# B&R Automation Studio project TD52 (part 46)

#### c_spare3Init.st
```iecst
(*******************************************************************************
CUSTOMIZED: c_spare3 			init to customized task placeholder

This code is confidential and proprietary to the INNIO Company.
It may not be used in any form, or reproduced in any manner,
without written permission of the INNIO Company.
Copyright, INNIO Company, 2019

Customized modifications: -
------------------------

Instructions for use:
--------------------
USE THIS TASK TO ADD CODE SNIPPETS AFTER ENGINE DELIVERY

Outstandings:
------------

*******************************************************************************)
PROGRAM _INIT

	bDoNothing := TRUE;

	(*-----------------------------------------------------------------------------*)
	bNoInitDetected := FALSE; 	 (* Insert this into every tasks INIT code to activate download detection *)
END_PROGRAM
```

### Program Logical/Customized/c_mns (IEC, version 4.14.0) - customisation task for grid power controller

#### c_mnsCyclic.st
```iecst
(*******************************************************************************
c_mns		 customizable mains demand controller  (derived from anf_nb 	customized engine demand depending of griddemand power setpoints)

This code is confidential and proprietary to the INNIO Company.
It may not be used in any form, or reproduced in any manner,
without written permission of the INNIO Company.
Copyright, INNIO Company, 2025

Customized modifications: -
------------------------

History:
-------
V4.04.1 14.11.2016 Zengerer			New task according to new spec. from Schwab Christoph, TPE (based on task anf_nb V4.03.0, 05.07.2013 pankayrodney)
V4.04.2 23.05.2017 Zengerer			Connect IN Interfaces to Hal tP_Mns_AnaIn, tDem_Ctr_Mns
V4.05.0 05.09.2017 zengerer			Nachziehen der Netzbezugsregler Änderungen von Schwab Christoph / Caks Michael aus File Bugs&Solution_MnsCtrl.zip
V4.05.1 30.11.2017 zengerer			50 + removed according to Basisupdate 4.4.0.6
V4.05.2 12.03.2018 zengerer			comments updated
V4.05.3 18.04.2018 Schwab Christoph bMsg2302_Enable-- bMsg2418_Enable Version
V4.05.4 20.04.2018 Zengerer			Timer Reset Button FUNCTION INVERTED; SOME UNTESTED CHANGES FROM V4.5.3 REVERTED
		25.04.2018 Zengerer			MM2VIS.rPmns_DemGenerate_Lim_On rPmns_DemGenerate_Lim_Off
V4.07.1 13.05.2019 Zengerer		 	Change of y_Min Y_Max strategy per option selection, ShadowPara_tCtr_Mns to prevent para writing; +activation Para
V4.11.0	24.02.2022 Perktold			impemented plant controller upgrade
V4.14.0	13.03.2025 Zengerer 		moved mains import controller activation bit

Instructions for use:
--------------------
 TASK REPLACES the task anf_nb. Do not activate anf_nb any more.

Outstandings:
------------
ADOPT ACCORDING TO PLANT SPECIFIC NEEDS

	-Testing for IN_CU.tP_Act[2].Ai has to be done
	-remove SparePara[73] V4.07 option here after testing phase
*******************************************************************************)
PROGRAM _CYCLIC

	(* IN INTERFACE: new V4.4.0,  2016 *)
	IN_CU.tDem_Ctr_Mns.Di	;				(*activation bit input (default value in case of not using interface moved to c_modIF) *)
	bDem_Ctr_Mns := IN_CU.tDem_Ctr_Mns.Di;  (*connect DI mns controller activation interface to hardware *)
	IN_CU.tP_Mns_AnaIn.Ai  ; 				(*AnaIn		Mains power Actual value over mA Signal *)
	IN_CU.tP_Mns_AnaIn.GoodQual ;			(*AnaIn		Mains power Actual value over mA Signal *)
	IN_CU.tP_Act[2].Ai;						(* P [kW] 	Mains power Actual value over MMU	*)

	IN_CU.rP_Nom;							(*Nominal power at selected gas type *)

	VIS2MM.tCtr_Mns_In;
//	VIS2MM.rPmns_setpoint ;					(* = p_MainsImport Setpoint *)
	IN_CU.tCtr_Mns_Anain_Setp_W_ext.Ai;		 (*AnaIn	Setpoint over mA Signal *)	//replaces:  = 	OUT_CU.rCustAnaIn[1] /100.0 ;
	IN_CU.tCtr_Mns_Anain_Setp_W_ext.GoodQual;(*AnaIn	Setpoint over mA Signal *)	//replaces:  = 	OUT_CU.rCustAnaIn[1] /100.0 ;

	Para.bCtr_Mns_Enable;				(*Parameter)	general activation bit for mns controller *)

	Para.tCtr_Mns.W_set;				(*Parameter	W(setpoint) start  Var.1:	internal setpoint *)
	Para.tCtr_Mns.W_min;				(*Parameter	W(setpoint) minimum *)
	Para.tCtr_Mns.W_max;				(*Parameter	W(setpoint) maximum *)
	Para.bCtr_Mns_AnaIn_Setp_Enable;	(*Parameter 	setpoint over mA aktiv Var.2: analog in setpoint *)
	Para.bCtr_Mns_Setp_Set4mA;			(*Parameter 	scaling 4-20 mA aktiv *)
	Para.rCtr_Mns_Setp_ScalMin;			(*Parameter 	scale minimum *)
	Para.rCtr_Mns_Setp_ScalMax;			(*Parameter 	scale maximum *)

	Para.bP_Mns_MMU_Enable;				(*Parameter 	TRUE = use MMU2 measurement reading, FALSE = use Analog Input reading from customer messurement euipment *)
	Para.bP_Mns_AnaIn_Enable := NOT Para.bP_Mns_MMU_Enable;		(*INTERNAL GENERATED HERE, necessary because bP_Mns_AnaIn_Enable is not a parameter on VIS anymore*)

	Para.bP_Mns_AnaIn_Set4mA;			(*Parameter 	value scaling 4-20 mA aktiv *)
	Para.rP_Mns_AnaIn_ScalMin;			(*Parameter 	scale minimum *)
	Para.rP_Mns_AnaIn_ScalMax;			(*Parameter 	scale maximum *)

	Para.bLimOnOff_aktiv;				(*Parameter)	TRUE = use mns-ctr output to perform engine demand on/off *)
	Para.rMainsImport_max;				(*Parameter)	Mains Import maximum warning limit	*)
	Para.rMainsImport_max_trip;			(*Parameter)	Mains Import maximum alarm limit *)
	Para.rMainsExport_max;				(*Parameter)	Mains Export maximum warning limit	*)
	Para.rMainsExport_max_trip;			(*Parameter)	Mains Export maximum alarm limit *)

	Para.rDemGenerate_Lim_On;			(*Parameter)	Grenzwert Einschaltung (% von PN Generator) *)
	Para.rTime_Dem_On_delay;			(*Parameter)	Delay time until engine demand on [sec] *)
	Para.rDemGenerate_Lim_Off;			(*Parameter)	Grenzwert Abschaltung (% von PN Generator) *)
	Para.rTime_Dem_Off_delay;			(*Parameter)	Delay time until engine demand off [sec]*)
	Para.tCtr_Mns.W_set;				(*Parameter)	W(setpoint) start *)

	(* OUT INTERFACE *)
	OUT_CU.bEngDSS_Mains  ;								(* == ANF_NB *)
	OUT_CU.rP_MainsImport ;				(* rP_MainsImport Interface to MM syncronising: +=grid to plant power value in [KW] *)
	OUT_CU.rP_Set_Mns_Norm;				(* engine power setpoint from grid controller out   *)

	MM2VIS.bEngDSS_Mains ;	// := OUT_CU.bEngDSS_Mains;	(* == ANF_NB *)
	MM2VIS.rPcsm_act ;					(* Consumer Power = p_MainsImport + rP_Act_Norm_Filt *)
	MM2VIS.rPmns_act ;		//:= OUT_CU.rP_MainsImport ;					(* p_MainsImport t (= OUT_CU.rP_MainsImpor) *)
	MM2VIS.rPmns_setpoint ;				(* selected p_MainsImport Setpoint, with ramps... *)
	MM2VIS.tCtr_Mns_Out;				(*Controler output structure for VIS*)
	MM2VIS.tCtr_Mns_Out.Active;			(*Controler output active*)
	MM2VIS.tCtr_Mns_Out.Y;				(* engine power etpoint from grid controller out   *)

	OUT_CU.tCtr_Mns_Out ;				(*Controler output structure *)
	OUT_CU.tCtr_Mns_In;					(*Copy of controler input structure for reuse in other modules *)

	(****************************************************************************************************)
	(*Calculation of power values*)
	//Mains Power set point import controller
	IF 	(*Para.bP_Mns_AnaIn_Enable*)Para.bCtr_Mns_AnaIn_Setp_Enable  AND IN_CU.tCtr_Mns_Anain_Setp_W_ext.GoodQual THEN // Schwab Ch. Falscher Parameter Angebunden	(*Parameter setpoint over mA aktiv Var.2:	Der Sollwert wird mittels externen mA Signal, welches über Parameter angepasst werden kann*)
		rP_Mains_Set := IN_CU.tCtr_Mns_Anain_Setp_W_ext.Ai;		(*AnaIn		Setpoint over mA Signal *)

	ELSE
	//	rP_Mains_Set := MM2VIS.tCtr_Mns_Out.W;			NEIN, GEHT hier SO NICHT mehr!	(* rP_GenerateSet		alt: 	soll_netz := REG1.w;*)
		rP_Mains_Set := Para.tCtr_Mns.W_set;  		(* rP_GenerateSet from Vis manual input	*)
	END_IF

	//Verbraucherleistung (= Netzbezugsleistung + Generatorleistung)
	rP_Consumption := rP_MainsImport + (IN_CU.rP_Act_Norm_Filt * IN_CU.rP_Nom);			(* verbrauch == rP_Consumption					alt: verbrauch := netzbezug + );*)

	(*Schwab Ch. => rP_DemGenerate wird immer berechnet! Keine IF Funktion benötigt*)
	rP_DemGenerate := rP_Consumption - rP_Mains_Set;
	MM2VIS.rPmns_DemGenerate := rP_DemGenerate;		(*new V4.5 beta *)

	(* P_MainsImport: measured absolute power from mains to plant in [KW] (+=grid to plant power, -=plant to grid*)	 //=Netzbezugsleistung
	IF 	Para.bP_Mns_MMU_Enable THEN 							(*Parameter TRUE = ISTwert Netzbezug über MMU gemessen (Var.2), 	FALSE = über mA Signal (Var.1)*)
		//FEHLT NOCH: NB- Leistung von eigenem MMU
		rP_MainsImport := 	IN_CU.tP_Act[2].Ai;					(* P [kW] Mains power Actual value over MMU	  := 98765.4321;		//FEHLT NOCH:  test  *)

	ELSIF  IN_CU.tP_Mns_AnaIn.GoodQual THEN 				(*AnaIn	Actual value mA Signal Quality Check*)
		rP_MainsImport := 	IN_CU.tP_Mns_AnaIn.Ai;		(*AnaIn	Istwert = über mA Signal (Var.1):	Der Istwert wird mittels mA Signal geliefert, welches über Parameter angepasst werden kann	 	alt: netzbezug := REAL_TO_INT(OUT_CU.rCustAnaIn[1]);	*)
	ELSE
		rP_MainsImport :=	(-rP_MainsImport_max) ;				(* failsafe value = no engine demand *)
	END_IF

	IF 	Para.bCtr_Mns_Enable AND bDem_Ctr_Mns THEN 	 (* TASK ACTIVATION by (Parameter)	Regler Aktivierung *)

		(* P_MainsImport_max limit parameter*)	//maximal erlaubte Netzbezugsleistung
	//	rP_MainsImport_max := DINT_TO_REAL(Para.rCust_SparePara[1]);		(*:= SPS_REZP1;				alt:netzbezug_max := INT_TO_UDINT(Para.rCust_SparePara[1]); *)
		rP_MainsImport_max :=  			Para.rMainsImport_max;				(*Parameter)	Mains Import maximum	alt:netzbezug_max := INT_TO_UDINT(Para.rCust_SparePara[1]); *)
						// old:			Para.rMainsImport_max_trip;			(*Parameter)	Mains Import maximum Abstellend True/False *)

		//Grenzwert [0-1 NOM Pnenn (früher %Pnenn!)] Anforderung EIN
		rP_DemGenerate_Lim_On :=		Para.rDemGenerate_Lim_On;			(*Parameter)	Grenzwert Einschaltung (% von PN Generator)  alt: p_ein_proz := INT_TO_UDINT( SPS_REZP1); *)

		//Grenzwert [0-1 NOM Pnenn (früher %Pnenn!)] Anforderung AUS
		rP_DemGenerate_Lim_Off :=		Para.rDemGenerate_Lim_Off;			(*Parameter)	Grenzwert Abschaltung (% von PN Generator) 	alt: p_aus_proz := INT_TO_UDINT( SPS_REZP2);*)

		//Nennleistung bei aktiver Gasart
		rP_Nom := (IN_CU.rP_Nom);					(*Nennleistung bei aktiver Gasart)  alt: zm := REAL_TO_INT(IN_CU.P_Nom);*)

		//Freigabe Netzbezugsregler
		//bDem_Ctr_Mns :=  ?  := bRSS_Rem AND IN_CU.bMCB_On AND IN_CU.GCB_ON AND IN_CU.AN_PGW1;		(*kann bRSS_Rem ersetzt werden durch bRSS_Rem? - nein *)
		OUT_CU.bEngDSS_Mains_Rel := IN_CU.bOMSS_Aut
								AND bRSS_Rem
								AND	IN_CU.bMCB_On
								AND Para.bCtr_Mns_Enable
								//	IN_CU.bGCB_On AND  NICHT einbinden, Regler kann sonst den motor nicht mehr starten!
								AND bDem_Ctr_Mns 	(*DI Customer Demand Input*)
								AND	(IN_CU.tP_Mns_AnaIn.GoodQual OR IN_CU.tP_Act[2].GoodQual);		(*lt. Schwab, 2017-11-28*)

		(*OUT_CU.bEngDSS_Mains_Block aktuell nicht in Verwendung => Wird über A2302 abgedeckt /  Schwab Ch.*)
		//		//Notabschaltung durch Überschreitung der erlaubten Rückspeiseleistung ins Netz (pb7/M_BLOCK)
//		xTOF_FA_BLOCK_NB.IN := (-rP_MainsImport) > rP_MainsImport_max;				(*shut down engine, if power to grid (=-MainsImport) exceeds allowed limt *)
//		xTOF_FA_BLOCK_NB.PT := REAL_TO_TIME(Para.rTime_Dem_Off_delay) * 1000;			(*Parameter)	[SEC] Zeitwert Verzögerung Abforderung alt: T#1m; *)
//		xTOF_FA_BLOCK_NB();
//
//		OUT_CU.bEngDSS_Mains_Block := xTOF_FA_BLOCK_NB.Q;

		//geforderte Generatorleistung (= Verbraucherleistung - Netzbezugsollwert)
//		IF bDem_Ctr_Mns THEN
//			rP_DemGenerate := MM2VIS.tCtr_Mns_Out.Y * rP_Nom; //Funktion doppelt? ->sonst TESTEN!
//		ELSE
//			rP_DemGenerate := rP_Consumption - rP_Mains_Set;					(*	soll_gen ==  rP_DemGenerate		alt: soll_gen := verbrauch - soll_netz; *)
//		END_IF

		//Berechnung Anforderungsleistung
//		zm1 := rP_DemGenerate_Lim_On * rP_Nom;				//Schwab remove: 50 + rP_DemGenerate_Lim_On * rP_Nom
////	zm1 := zm1/100;
//		p_ein := (zm1);												(*UDINT_TO_INT(zm1);*)
		p_ein := rP_DemGenerate_Lim_On * rP_Nom;			//Schwab remove: 50 + rP_DemGenerate_Lim_On * rP_Nom
		MM2VIS.rPmns_DemGenerate_Lim_On := p_ein;		(*new V4.5 beta *)

		//Berechnung Abwahlleistung
//		zm0 := rP_DemGenerate_Lim_Off * rP_Nom;				//Schwab remove: 50 + rP_DemGenerate_Lim_Off * rP_Nom
////	zm0 := zm0/100;
//		p_aus := (zm0);												(*UDINT_TO_INT(zm0);*)
		p_aus := rP_DemGenerate_Lim_Off * rP_Nom;			//Schwab remove: 50 + rP_DemGenerate_Lim_Off * rP_Nom
		MM2VIS.rPmns_DemGenerate_Lim_Off := p_aus;		(*new V4. beta5 *)

		//Anforderung EIN
		IF AUS AND NOT bDisplayTimerHelper THEN
			TON_R_MnsDemandOn.PT := REAL_TO_UDINT(Para.rTime_Dem_On_delay) * 100;
		END_IF
		TON_R_MnsDemandOn(IN := (rP_DemGenerate >= p_ein));				(*caution, RS will NOT WORK here as intended! *)
	//	TON_R_MnsDemandOn(IN := (rP_DemGenerate >= p_ein), PT := 	(Para.tiTime_Dem_On_delay) * 1000, RS := VIS2MM.bTime_Dem_On_delay_Reset);
		IF VIS2MM.bTime_Dem_On_delay_Reset	THEN		(*IF VIS Timer Reset Button is pressed*)
			VIS2MM.bTime_Dem_On_delay_Reset := FALSE;	(*clear button*)
			TON_R_MnsDemandOn( PT := 0 );				(*runout timer*)
			TON_R_MnsDemandOff( PT := 0 );				(*runout timer*)
			bDisplayTimerHelper := TRUE;				(*Visu helper bit for TON_R_MnsDemandOn display*)
		END_IF
		IF (IN_CU.rN_EngAct > 450) AND (IN_CU.rN_EngAct < 750) THEN 	bDisplayTimerHelper := FALSE; END_IF			(*Reset Visu helper bit for TON_R_MnsDemandOn display*)

		EIN := TON_R_MnsDemandOn.Q;
		MM2VIS.rTime_Dem_On_CntDn := UDINT_TO_REAL(TON_R_MnsDemandOn.PT - TON_R_MnsDemandOn.ET) /100 ;		(* Display start count down *)
	//	MM2VIS.tiTime_Dem_On_CntDn := 			  (TON_R_MnsDemandOn.PT - TON_R_MnsDemandOn.ET) /1000 ;		(* Display start count down *)

		//Anforderung AUS
		IF EIN AND NOT bDisplayTimerHelper THEN
			TON_R_MnsDemandOff.PT := REAL_TO_UDINT(Para.rTime_Dem_Off_delay) * 100; 	(*Parameter)	Delay time until engine demand off [sec]*)
			MM2VIS.rTime_Dem_On_CntDn := UDINT_TO_REAL(TON_R_MnsDemandOff.PT - TON_R_MnsDemandOff.ET) /100 ;		(* Display start count down *)
		END_IF
		TON_R_MnsDemandOff(IN := (rP_DemGenerate <= p_aus));		(* PREPARED for AUS := soll_gen <= p_aus;*)
		AUS := 	TON_R_MnsDemandOff.Q;
	//	AUS := rP_DemGenerate <= p_aus;								(* := soll_gen <= p_aus;*)

		//Anforderung
		OUT_CU.bEngDSS_Mains := (EIN OR OUT_CU.bEngDSS_Mains)
							AND NOT AUS			(* OUT_CU.bEngDSS_Mains == ANF_NB *)
							AND Para.bLimOnOff_aktiv;

		(*Connection failure bit for message set*)
		(* A2302 mains export power limit: Shut down engine, if NEGATIVE Mains Import (= power export to the grid) is exceeding (<) the allowed limit (-Limit value)  *)
		bMsg2302_Enable	:=	Para.bCtr_Mns_Enable
//						AND Para.bLimOnOff_aktiv 				// gehört nicht zu dieser Funktion / Schwab Ch.
						AND ((*IN_CU.tDem_Ctr_Mns.Di*)bDem_Ctr_Mns OR Para.iCtr_Mns_Options.2);

		bMsg2302_Set	:=	OUT_CU.rP_MainsImport < (-Para.rMainsExport_max_trip);

		(* A2303 mains import controller limit 2  ??? Why shut down the engine, if too few power is available  ???	*)
		bMsg2303_Enable	:=	Para.bCtr_Mns_Enable
//						AND Para.bLimOnOff_aktiv 				// gehört nicht zu dieser Funktion / Schwab Ch.						AND Para.bLimOnOff_aktiv
						AND (*IN_CU.tDem_Ctr_Mns.Di*)bDem_Ctr_Mns
						AND ((*IN_CU.tDem_Ctr_Mns.Di*)bDem_Ctr_Mns OR Para.iCtr_Mns_Options.3) 			(*Change 2018 Ze: Alarm only active in Ctr_Mns mode (using option bit 3 and 4 of INTERNAL parameter, ->NORMALY SWITCHED TO FALSE*)
						AND Para.iCtr_Mns_Options.4
						AND FALSE;	// Funktion muss nochmals mit betroffene Personen diskutiert werden / Schwab Ch.

		bMsg2303_Set	:= OUT_CU.rP_MainsImport > Para.rMainsImport_max_trip;

		(* W2415 mains import controller: Messsignalstörung Netzbezugs- Sollwert 	*)
		bMsg2415_Enable	:=	Para.bCtr_Mns_Enable
						AND Para.bCtr_Mns_AnaIn_Setp_Enable
						AND (IN_CU.tDem_Ctr_Mns.Di OR Para.iCtr_Mns_Options.5);	(*Change 2018 Ze: Alarm only active in Ctr_Mns mode (using option bit 5 and 4 of INTERNAL parameter, ->NORMALY SWITCHED TO FALSE*)

		bMsg2415_Set	:= NOT IN_CU.tCtr_Mns_Anain_Setp_W_ext.GoodQual;

		(* W2416 mains import controller: Messsignalstörung Netzbezugs- Istwert	*)
		bMsg2416_Enable	:=	Para.bCtr_Mns_Enable
						AND	bDem_Ctr_Mns
						AND Para.bP_Mns_AnaIn_Enable
						AND Para.bP_Mns_AnaIn_Set4mA
						AND ((*IN_CU.tDem_Ctr_Mns.Di*)bDem_Ctr_Mns OR (NOT Para.iCtr_Mns_Options.6));

		bMsg2416_Set	:= NOT IN_CU.tP_Mns_AnaIn.GoodQual;

		(* W2417 mains export power limit: Warning, if NEGATIVE Mains Import (= power export to the grid) is exceeding (<) the allowed limit (-Limit value)  *)
		bMsg2417_Enable	:=	Para.bCtr_Mns_Enable  					//AND Para.bLimOnOff_aktiv;
						AND bDem_Ctr_Mns
						AND ((*IN_CU.tDem_Ctr_Mns.Di*)bDem_Ctr_Mns OR (NOT Para.iCtr_Mns_Options.7));

		bMsg2417_Set	:= OUT_CU.rP_MainsImport < (-Para.rMainsExport_max) ;

		(* W2418  mains import controller limit 2:  Warning if positive Mains Import (= power drawn from the grid) is exceeding (>) the allowed limit (+Limit value)*)
		bMsg2418_Enable	:=	Para.bCtr_Mns_Enable 					//AND Para.bLimOnOff_aktiv AND FALSE;
						AND bDem_Ctr_Mns
						AND ((*IN_CU.tDem_Ctr_Mns.Di*) bDem_Ctr_Mns OR Para.iCtr_Mns_Options.8);

		bMsg2418_Set	:= OUT_CU.rP_MainsImport > Para.rMainsImport_max;

	ELSE
		//Task disabeled, keine Anforderung
		bMsg2302_Enable		 		:= FALSE;
		bMsg2302_Set		 		:= FALSE;
		bMsg2303_Enable		 		:= FALSE;
		bMsg2303_Set		 		:= FALSE;
		bMsg2415_Enable		 		:= FALSE;
		bMsg2415_Set		 		:= FALSE;
		bMsg2416_Enable		 		:= FALSE;
		bMsg2416_Set		 		:= FALSE;
		bMsg2417_Enable		 		:= FALSE;
		bMsg2417_Set		 		:= FALSE;
		bMsg2418_Enable		 		:= FALSE;
		bMsg2418_Set		 		:= FALSE;
		OUT_CU.bEngDSS_Mains 		:= FALSE;
		OUT_CU.bEngDSS_Mains_Rel	:= FALSE;

	END_IF

	(******************************************************************************)
	(* MAINS POWER IMPORT/EXPORT CONTROLLER [kW] (System 1 from Lettenbichler- Plant Control) *)
//	IF 	Para.bCtr_Mns_Enable  THEN 	 (* ACTIVATION by (Parameter)  V4.07:  integratet in .enable *)
		(* PlantOperMode = 1 *)
		VIS2MM.tCtr_Mns_In.enable   	:= 	OUT_CU.bEngDSS_Mains_Rel AND Para.bCtr_Mns_Enable ; //bDem_Ctr_Mns ;		(*(Schnittstelle)	Aktivierung über Kundenschnittstelle *)
		VIS2MM.tCtr_Mns_In.W_ext    	:=  rP_Mains_Set;  				(*	Setpoint over mA Signal  FEHLT NOCH: .w_ref    := MAX (IN_MC.ENG_nom[1].Pgen, Pgen_dmnd_nom);(* reference value, units like "x" *)
		VIS2MM.tCtr_Mns_In.W_ext_Active := 	Para.bCtr_Mns_AnaIn_Setp_Enable ;		(* setpoint activation,  old: Para.Pmns_sp;  *)

		VIS2MM.tCtr_Mns_In.W_set2_Active	:= FALSE;	(*Input to define which internal setpoint will be used TRUE = use the 2nd set point | FALSE use the normal "1st" one*)
		VIS2MM.tCtr_Mns_In.GainScheduling	:= 0.0;		(*Input for Gain Scheduling: 0.0 = use 100% of the Standard PID-Parameters | 1.0 = use 100% of the GainSched. PID Parameters | linear interpolation in between*)
		VIS2MM.tCtr_Mns_In.Y_min_cust;					(*"customized" Y-Min at the current moment (The existing Y-Min parameter is the global minimum. To have an effect Y_min_cust needs to be > the parameter | -1.0 = function not used*)
		VIS2MM.tCtr_Mns_In.Y_max_cust;					(*"customized" Y-Max at the current moment (The existing Y-Max parameter is the global maximum. To have an effect Y_max_cust needs to be < the parameter | 1.0 = function not used*)
		VIS2MM.tCtr_Mns_In.Retrigger;					(*a rising edge on this input signals the controller to retrigger - set W on X and force the Integrator to the current Y*)
		VIS2MM.tCtr_Mns_In.A;							(*feed forward Input*)

		VIS2MM.tCtr_Mns_In.X			:= rP_MainsImport;				(* actual value, "PV Name" of "x" *)

		//	VIS2MM.tCtr_Mns_In.mode     	:= 1;   	     		     	(* 1: dy=Ki*(w-x/w_ref), 0: dy=Ki *)

		Para.tCtr_Mns.deadband	;  // 	:= 10.0;				(* dead band, units like "x" *)
		IF Para.tCtr_Mns.Tn = 0 THEN Para.tCtr_Mns.Tn := 110; END_IF // VIS2MM.tCtr_Mns_In.Ki_plus  := Speed_P_Ad/10;	(* units "In"/100ms=task class *)
									 Para.tCtr_Mns.Tn  ; 			 // VIS2MM.tCtr_Mns_In.Ki_minus := Speed_P_Ad/10;	(* units "In"/100ms=task class *)
		IF Para.tCtr_Mns.dY_max = 0 THEN Para.tCtr_Mns.dY_max := 0.1;	END_IF			(*  *)
		Para.tCtr_Mns.Y_block  	;	//:= 1.0;				(* % *)

		Para.tCtr_Mns.invert   ; 		//  := TRUE;			 	(* FALSE: x>w: decrease y, TRUE: x>w: increase y *)

		(*Beginn V4.07 change *)
		ShadowPara_tCtr_Mns			:= Para.tCtr_Mns;	(* controler internal derouting of para *)

		rY_min	:= LIMIT( (IN_CU.rP_Act_Norm_Filt - 0.03), (IN_CU.rP_Set_Min_Norm -0.03), 1.0);
		rY_max	:= LIMIT( (IN_CU.rP_Act_Norm_Filt + 0.03),  IN_CU.rP_Set_Min_Norm       , 1.0);
		bOptParaChangeAllowed := Para.rCust_SparePara[73] > 0;		(*V4.07 Bugfix disabeling, to allow temporary switch back to V4.05 behavior  *)
		IF bOptParaChangeAllowed  AND Para.bCtr_Mns_Enable THEN		(*V4.07 Change of y_Min Y_Max strategy per option selection, to prevent para writing *)
			Para.tCtr_Mns.Y_min	:= 	rY_min;		(* change, this is not allways possible! Caution, watch this LIMIT(Mn, IN, MX) para order to used functions priority handling of MN *)
			Para.tCtr_Mns.Y_max	:= 	rY_max;
		END_IF
//			VIS2MM.tCtr_Mns_In.Y_set := LIMIT(0.5,( LIMIT(rY_min, OUT_CU.tCtr_Mns_Out.Y, rY_max) ), 1.0);				(*test: Y limit without para change*)
//			VIS2MM.tCtr_Mns_In.Y_set_Active := (rY_min > OUT_CU.tCtr_Mns_Out.Y) OR (rY_max < OUT_CU.tCtr_Mns_Out.Y); 	(*test: Y limit without para change*)
			IF NOT VIS2MM.tCtr_Mns_In.enable THEN 			(* IF stopped controller THEN move internal y limit following actual set power (ELSE use Para. values) *)
				ShadowPara_tCtr_Mns.Y_min	:= rY_min; //:=	LIMIT(0.5, rY_min, 1);	(* controler internal derouting of para *)
				ShadowPara_tCtr_Mns.Y_max	:= rY_max; //:=	LIMIT(0.5, rY_max, 1);	(* controler internal derouting of para *)
			END_IF

		(*End V4.07 change *)

		OUT_CU.tCtr_Mns_In	:=	VIS2MM.tCtr_Mns_In;
		OUT_CU.tCtr_Mns_Out	:=	MM2VIS.tCtr_Mns_Out;

			xGeACtr_Mns;		(*Controller- FUNCTION CALL*)

	//	rP_DemGenerate 			:= MM2VIS.tCtr_Mns_Out.Y;	 	//Funktion doppelt? ->sonst TESTEN! (* "PV Name" of "y", % *)
		OUT_CU.rP_MainsImport :=	rP_MainsImport;					(*Interface to MM syncronising: +=grid to plant power value in [KW], -=plant to grid power*)
		OUT_CU.rP_Set_Mns_Norm	:= MM2VIS.tCtr_Mns_Out.Y;
		MM2VIS.rP_DemGenerate := rP_DemGenerate;
		MM2VIS.bEngDSS_Mains := OUT_CU.bEngDSS_Mains;	(* == ANF_NB *)
		MM2VIS.rPcsm_act := rP_Consumption;				(* Consumer Power = p_MainsImport + rP_Act_Norm_Filt *)
		MM2VIS.rPmns_act := OUT_CU.rP_MainsImport ;		(* p_MainsImport t (= OUT_CU.rP_MainsImpor) *)
		MM2VIS.rPmns_setpoint := rP_Mains_Set;			(*Actual main import power set point*)

//	END_IF

	//<outdated variants removed>

END_PROGRAM
```

#### c_mnsInit.st
```iecst
(*******************************************************************************
c_mns INIT		 customizable mains demand controller

This code is confidential and proprietary to the INNIO Company.
It may not be used in any form, or reproduced in any manner,
without written permission of the INNIO Company.
Copyright, INNIO Company, 2022

*******************************************************************************)
PROGRAM _INIT
	IF rP_MainsImport_max = 0 THEN rP_MainsImport_max := 999999; END_IF

	Para.bCtr_Mns_Enable;		(*Parameter)	Regler Aktivierung *)
	Para.tCtr_Mns.W_set;		(*Parameter	W(setpoint) start  Var.1:	Der Sollwert wird mittels wird über einen internen Parameter (Setpoint) realisiert *)
	Para.tCtr_Mns.W_min;		(*Parameter	W(setpoint) minimum *)
	Para.tCtr_Mns.W_max;		(*Parameter	W(setpoint) maximum *)

	Para.bCtr_Mns_AnaIn_Setp_Enable;(*Parameter 	setpoint over mA aktiv Var.2:	Der Sollwert wird mittels externen mA Signal, welches über Parameter angepasst werden kann*)
	Para.bCtr_Mns_Setp_Set4mA;		(*Parameter 	scaling 4-20 mA aktiv *)
	Para.rCtr_Mns_Setp_ScalMin;		(*Parameter 	scale minimum *)
	Para.rCtr_Mns_Setp_ScalMax;		(*Parameter 	scale maximum *)

	Para.bP_Mns_MMU_Enable;			(*Parameter 	FALSE = über mA Signal Var.1:	Der Istwert wird mittels mA Signal, welches über Parameter angepasst werden kann *)
	Para.bP_Mns_AnaIn_Set4mA;		(*Parameter 	scaling 4-20 mA aktiv *)
	Para.rP_Mns_AnaIn_ScalMin;		(*Parameter 	scale minimum *)
	Para.rP_Mns_AnaIn_ScalMax;		(*Parameter 	scale maximum *)

	Para.bLimOnOff_aktiv;			(*Parameter)	Regler Aktivierung		*)
	Para.rMainsImport_max;			(*Parameter)	Mains Import maximum	*)
	Para.rMainsImport_max_trip;		(*Parameter)	Mains Import maximum Abstellend True/False *)
	Para.rMainsExport_max;			(*Parameter)	Mains Export maximum	*)
	Para.rMainsExport_max_trip;		(*Parameter)	Mains Export maximum Abstellend True/False *)
	Para.rDemGenerate_Lim_On;		(*Parameter)	Grenzwert Einschaltung (% von PN Generator) *)
	Para.rTime_Dem_On_delay;		(*Parameter)	Zeitwert Verzögerung Anforderung *)
	Para.rDemGenerate_Lim_Off;		(*Parameter)	Grenzwert Abschaltung (% von PN Generator) *)
	Para.rTime_Dem_Off_delay;		(*Parameter)	Zeitwert Verzögerung Abforderung *)

	Para.rTime_Trip_MainsImort;		(*ALT! Parameter)	Verzögerung Abstellung bei Überschreitung *)
	Para.rTime_Trip_MainsExport;	(*ALT! Parameter)	Verzögerung Abstellung bei Überschreitung *)

	(*Supply defaults for missing/not used VIS parameter*)
	ParaFactoryDefault.tCtr_Mns.W_set := 123.4;
	ParaFactoryDefault.tCtr_Mns.W_min := 0.0;
	ParaFactoryDefault.tCtr_Mns.W_max := 88888.8;
	ParaFactoryDefault.tCtr_Mns.dW_up := 0.1;
	ParaFactoryDefault.tCtr_Mns.dW_down := 0.1;
	ParaFactoryDefault.tCtr_Mns.deadband := 3.0;
	ParaFactoryDefault.tCtr_Mns.Y_min := 0.5;
	ParaFactoryDefault.tCtr_Mns.Y_max := 1.0;
	ParaFactoryDefault.tCtr_Mns.Y_block  := 1.0;
	ParaFactoryDefault.tCtr_Mns.Kp := 0.01;
	ParaFactoryDefault.tCtr_Mns.Tn := 150.0;
	ParaFactoryDefault.tCtr_Mns.Tv := 0.0;

	ParaFactoryDefault.tCtr_Mns.t_min_pulse_up := 0.20;
	ParaFactoryDefault.tCtr_Mns.t_period_up := 1.0;
	ParaFactoryDefault.tCtr_Mns.t_min_pulse_down := 0.2;
	ParaFactoryDefault.tCtr_Mns.t_period_down := 1.0;
	ParaFactoryDefault.tCtr_Mns.invert := TRUE ;

	(* configure and asign structures for mains input controller *)
//	xGeACtr_Mns(pParameter := ADR(Para.tCtr_Mns), 		pInput := ADR(VIS2MM.tCtr_Mns_In), pOutput := ADR(MM2VIS.tCtr_Mns_Out));
	xGeACtr_Mns(pParameter := ADR(ShadowPara_tCtr_Mns),	pInput := ADR(VIS2MM.tCtr_Mns_In), pOutput := ADR(MM2VIS.tCtr_Mns_Out));  (* V4.07 *)

	VIS2MM.tCtr_Mns_In.AlwaysUseYRamp		:= TRUE;	(*If TRUE the Y signal will always limit the change rate via the according parameter | if FALSE the Y signal will jump in case the controller is disabled (blocked or set)*)
	VIS2MM.tCtr_Mns_In.KeepYManAtBlock		:= TRUE;	(*If TRUE the controller will keep the Y-man value constant in case the controller is disabled (blocked or set) | If FALSE the blocked or set value will override the Y-man value*)
	VIS2MM.tCtr_Mns_In.Y_min_cust			:= -1.0;	(*"customized" Y-Min at the current moment (The existing Y-Min parameter is the global minimum. To have an effect Y_min_cust needs to be > the parameter | -1.0 = function not used*)
	VIS2MM.tCtr_Mns_In.Y_max_cust			:=  1.0;	(*"customized" Y-Max at the current moment (The existing Y-Max parameter is the global maximum. To have an effect Y_max_cust needs to be < the parameter | 1.0 = function not used*)
	VIS2MM.tCtr_Mns_In.StepperMode			:= FALSE;	(* TRUE = use PWM-Mode (standard mode until 4.10) | FALSE = use continuous servo drive *)

END_PROGRAM
```

#### c_mns.var
```iecst
VAR
	xGeACtr_Mns : GeACtr;
	rP_Mains_Set : REAL; (* Sollwert Netzbezugsregler *)
	p_ein : REAL; (* Anforderungsleistung *)
	p_aus : REAL; (* Abwahlleistung *)
	rP_Consumption : REAL; (* Verbraucherleistung *)
	rP_DemGenerate : REAL; (* Geforderte Generatorleistung *)
	rP_MainsImport_max : REAL; (* max. erlaubte Netzbezugsleistung absolut [KW]*)
	rP_MainsImport : REAL; (* Netzbezugsleistung absolut [KW]*)
	rP_DemGenerate_Lim_Off : REAL; (*Ausschaltlimit in % Pn*)
	rP_DemGenerate_Lim_On : REAL; (*Einschaltlimit in % Pn*)
	rP_Nom : REAL;
	EIN : BOOL; (*release engine start*)
	AUS : BOOL; (*release engine stop*)
	TON_R_MnsDemandOn : TON_R := (0);
	TON_R_MnsDemandOff : TON_R := (0); (*V4.5 prepared*)
	bDem_Ctr_Mns : BOOL := 0;
	bDisplayTimerHelper : BOOL; (*Visu helper bit for TON_R_MnsDemandOn display*)
	rY_min : REAL; (*temporary limiting y*)
	rY_max : REAL; (*temporary limiting y*)
	bOptParaChangeAllowed : BOOL := FALSE; (*TRUE will allow programmable changes of Y_Min and Y_Max parameter values*)
	ShadowPara_tCtr_Mns : _tGeACtrPara; (*TASK INTERNAL working copy with adopted limit values *)
END_VAR
```

### Program Logical/Customized/anf_nb (IEC, version 4.03.0) - customisation task for grid power controller

#### anf_nbCyclic.st
```iecst
(*******************************************************************************
anf_nb 			customized engine demand depending of griddemand power setpoints

This code is confidential and proprietary to the INNIO Company.
It may not be used in any form, or reproduced in any manner,
without written permission of the INNIO Company.
Copyright, INNIO Company, 2019

Customized modifications: -
------------------------

History:
-------
V3.90.0	??-??-2012 ?pankayrodney?  	converted from LD
V3.90.1	14-12-2012 Zengerer			rework, renaming of some varnames according to naming convention
V3.91	14.02.2013 zengerer			datatypes changed to real...
V3.92	05.07.2013 zengerer			new interface OUT_CU.rP_MainsImport
V4.03.0	05.07.2013 zengerer			Bugfix: remove predefined reserve parameter numbers to avoid unintended task activation
!ALT! TASK NICHT MEHR VERWENDEN- - -> c_mns

Instructions for use:
--------------------
OUT_CU.bEngDSS_Mains  (==ANF_NB) generated depending on utility demand signals

Outstandings:
------------
!ALT! TASK NICHT MEHR VERWENDEN- - -> c_mns

*******************************************************************************)
PROGRAM _INIT

	(*	OLD TASK - DO NOT USE ANYMORE! *)

	(*Functionality MOVED TO TASK c_mms *)

END_PROGRAM
```

### Program Logical/Customized/c_statGR (IEC, version 4.09.0) - customisatio task for static GridCode functions

#### c_statGRCyclic.st - Cyclic code
```iecst
(*********************************************************************************************
AGGR: static GridCode - custom task (cyclic)

This code is confidential and proprietary to the INNIO Company.
It may not be used in any form, or reproduced in any manner, without the express
written permission of the INNIO Company.
Copyright, INNIO Company, 2019

- Auftragsspzifische Anpassungen für das stat. GridCode Paket

Customized modifications: -
------------------------

History:
-------
V3.40.0	14-02-2013	Perktold,  generated
V3.40.1	12-06-2013	Perktold,  user-friendliness-upgrade
V4.00.0 22-08-2013  Maxhera,   implementation of the module for modular software
V4.03.0 13-01-2016	Perktold,  changed for use in MM Customized
V4.04.0	06-10-2016	Perktold,  changed ERDF/DEIE - Activation now via Parameter
V4.04.0	02-11-2016	Gwiggner,  added frequency control
V4.05.0 01-12-2017  Farre, 	   added/modified Q functions, Point of control/reference, P(U)
V4.05.0 04-12-2017	lettenb.   GR: custom measurement POC(point of control)added
                               tProtectionTest[x].Do added, grid code logic
V4.06.0 06-08-2018  Zuschnig   added signal loss function for P_Set, P_Lim, COSPHI_Set, Q_Set, Q_Lim and U_Set
V4.07.0 15-01-2019	Zuschnig,  Added Parameter von AI oder BUS
V4.09.0 28.11.2019	lettenb.   protection test moved to separate task
V4.13.0	12.10.2023	Farre,	   added ILF (de)activating HW, Bus and feedback signals

Instructions for use:
--------------------
-
Outstandings:
-------------
*********************************************************************************************)

PROGRAM _CYCLIC
(********************************************************************************************)
(* TASKAUFBAU: ==>	 TASK STRUCTURE															*)
(*																							*)
(* A) BLINDLEISTUNG ==>	  REACTIVE POWER													*)
(*	o cos(phi) - Sollwertvorgabe ==> cos(phi) Setpoint										*)
(*	o Q - Sollwertvorgabe																	*)
(*	o Q - Limitierung																		*)
(*	o cos(phi) = f(P)																		*)
(*	o U - Sollwert (für Q(U) & cos(phi)=f(U) notwendig)	/ U control  						*)
(*	o Q(U)																					*)
(*	o cos(phi) = f(U)																		*)
(*	o Q = f(P)																				*)
(*	o Priorisierung der Funktionen (notwendig wenn mehr als eine verwendet werden)			*)
(*	o Analogausgänge																		*)
(*	o Point of reference - Customized														*)
(*	o Point of control - Customized													    	*)
(*	o Reactive Power control function - Customized											*)
(*																							*)
(* B) WIRKLEISTUNG																			*)
(*	o Sollwertvorgabe																		*)
(*	o Leistungslimitierung																	*)
(*	o PFC - PrimaryFrequencyControl															*)
(*	o RMC - RegulatingMarginControl															*)
(*																							*)
(*	o P(U) - Österreich																		*)
(********************************************************************************************)

(********************************************************************************************)
(*************** B L I N D L E I S T U N G ** / ** R E A C T I V E   P O W E R **************)
(********************************************************************************************)

(********************************************************************************************)
(********************** COS (PHI) - S E T P O I N T  S E L E C T I O N **********************)
(********************************************************************************************)
	(*(DE)Activating  - HW --> To connect or to set fix value    			         			*)
	OUT_CU.bPF_GenC_SetEUCOn 	:= IN_CU.tPF_GenC_SetEUCOn.Di; 			(*DI:setpoint genetaror power factor(COS PHI)from EU - on(activate)   *)
	OUT_CU.bPF_GenC_SetEUCOf 	:= IN_CU.tPF_GenC_SetEUCOf.Di := TRUE; 	(*DI:setpoint genetaror power factor(COS PHI)from EU - off(deactivate)*)

	(* Marshalling DI: COSPHI-fixed values to the individual steps       		        		*)
	OUT_CU.PF_GenC_SetFix1	:= IN_CU.tPF_GenC_SetFix1EU.Di;	(*DI: setpoint genetaror power factor(COS PHI) - Fixvalue 1 from EU *)
	OUT_CU.PF_GenC_SetFix2	:= IN_CU.tPF_GenC_SetFix2EU.Di;	(*DI: setpoint genetaror power factor(COS PHI) - Fixvalue 2 from EU *)
	OUT_CU.PF_GenC_SetFix3	:= IN_CU.tPF_GenC_SetFix3EU.Di;	(*DI: setpoint genetaror power factor(COS PHI) - Fixvalue 3 from EU *)
	OUT_CU.PF_GenC_SetFix4	:= IN_CU.tPF_GenC_SetFix4EU.Di;	(*DI: setpoint genetaror power factor(COS PHI) - Fixvalue 4 from EU *)
	OUT_CU.PF_GenC_SetFix5	:= IN_CU.tPF_GenC_SetFix5EU.Di;	(*DI: setpoint genetaror power factor(COS PHI) - Fixvalue 5 from EU *)

	(*(DE)activation - bus          		         					                        *)
	OUT_CU.bGenC_PFBC_SetCOn;				(*bus: setpoint  genetaror power factor (COS PHI) from EU - on (activate)*)
	OUT_CU.bGenC_PFBC_SetCOf 	:= TRUE;	(*bus: setpoint  genetaror power factor (COS PHI) from EU - off (deactivate)*)

	(* connection bus signal - COS(PHI) set value from EU                                       *)
	(* to do:																		        	*)
	(* - BusSetpoint OUT_CU.rGenC_PFBC              				 		                    *)
	(* - bPFBC_GenC_SetErrBC generate - if TRUE it will be used Backupvale (Parameter)          *)
	OUT_CU.rGenC_PFBC;			(*bus: signal value genetaror power factor (COS PHI) from EU [-]*)
	OUT_CU.bPFBC_GenC_SetErrBC;	(*bus: setpoint generator power factor (COS PHI) from EU error - use backupvalue*)

	(*- - - - - - - - - - - - - - - - -  F E E D B A C K  S I G N A L S  - - - - - - - - - - -  *)
	IN_CU.tPF_GenC_SOn.Do;      (* generator power factor (COS PHI) from EU is on               *)
	IN_CU.tPF_GenC_SOf.Do;      (* generator power factor (COS PHI) from EU is off              *)
	IN_CU.tPF_GenC_Fix1SOn.Do;	(* genetaror power factor (COS PHI) - fixvalue 1 from EU is on  *)
	IN_CU.tPF_GenC_Fix2SOn.Do;	(* genetaror power factor (COS PHI) - fixvalue 2 from EU is on  *)
	IN_CU.tPF_GenC_Fix3SOn.Do;	(* genetaror power factor (COS PHI) - fixvalue 3 from EU is on  *)
	IN_CU.tPF_GenC_Fix4SOn.Do;	(* genetaror power factor (COS PHI) - fixvalue 4 from EU is on  *)
	IN_CU.tPF_GenC_Fix5SOn.Do;	(* genetaror power factor (COS PHI) - fixvalue 5 from EU is on  *)
	(********************************************************************************************)

	(********************************************************************************************)
	(************************** Q - S E T P O I N T  S E L E C T I O N **************************)
	(********************************************************************************************)
	(*(DE)Activating  - HW --> To connect or to set fix value    		         			    *)
	OUT_CU.bQ_GenC_SetEUCOn		:= IN_CU.tQ_GenC_SetEUCOn.Di;		(*DI: setpoint reactive power characteristic (Q) from EU - on (activate)   *)
	OUT_CU.bQ_GenC_SetEUCOf 	:= IN_CU.tQ_GenC_SetEUCOf.Di:=TRUE;	(*DI: setpoint reactive power characteristic (Q) from EU - off (deactivate)*)

	(*Marshalling DI: Q fixed values to the individual steps									*)
	OUT_CU.Q_GenC_SetFix1		:= IN_CU.tQ_GenC_SetFix1EU.Di;	(*DI: reactive power (Q) - Q-fixvalue 1 from EU	*)
	OUT_CU.Q_GenC_SetFix2		:= IN_CU.tQ_GenC_SetFix2EU.Di;	(*DI: reactive power (Q) - Q-fixvalue 2 from EU	*)
	OUT_CU.Q_GenC_SetFix3		:= IN_CU.tQ_GenC_SetFix3EU.Di;	(*DI: reactive power (Q) - Q-fixvalue 3 from EU	*)
	OUT_CU.Q_GenC_SetFix4		:= IN_CU.tQ_GenC_SetFix4EU.Di;	(*DI: reactive power (Q) - Q-fixvalue 4 from EU	*)
	OUT_CU.Q_GenC_SetFix5		:= IN_CU.tQ_GenC_SetFix5EU.Di;	(*DI: reactive power (Q) - Q-fixvalue 5 from EU	*)

	(*(DE)Activating  - bus          		         					                       	*)
	OUT_CU.bGenC_QBC_SetCOn;			(* bus: setpoint reactive power (Q) from EU - on (activate)	       *)
	OUT_CU.bGenC_QBC_SetCOf	:= TRUE;	(* bus: setpoint reactive power (Q) from EU - off (deactivate)	   *)

	(* BUSSIGANAL connection  - Q set value from EU                                             *)
	(* to do:																					*)
	(* - BusSetpoint OUT_CU.rGenC_QBC              				 		                    	*)
	(*  - OUT_CU.bQ_GenC_SetErrBC generieren - falls TRUE wird der Backupwert (Parameter) verwendet		*)
	OUT_CU.rGenC_QBC;       	(* bus: scaling value reactive power (Q) from EU [kVAr]					*)
	OUT_CU.bQ_GenC_SetErrBC;	(* bus: Q setpoint BUS EU error - use backupvalue						*)

	(*- - - - - - - - - - - - - - - - -  F E E D B A C K  S I G N A L S  - - - - - - - - - - -  *)
	IN_CU.tQ_GenC_SOn.Do;     (* reactive power characteristic (Q) from EU is on  *)
	IN_CU.tQ_GenC_SOf.Do;     (* reactive power characteristic (Q) from EU is off *)
	IN_CU.tQ_GenC_Fix1SOn.Do; (* reactive power (Q) - Q-fixvalue 1 from EU on     *)
	IN_CU.tQ_GenC_Fix2SOn.Do; (* reactive power (Q) - Q-fixvalue 2 from EU on     *)
	IN_CU.tQ_GenC_Fix3SOn.Do; (* reactive power (Q) - Q-fixvalue 3 from EU on     *)
	IN_CU.tQ_GenC_Fix4SOn.Do; (* reactive power (Q) - Q-fixvalue 4 from EU on     *)
	IN_CU.tQ_GenC_Fix5SOn.Do; (* reactive power (Q) - Q-fixvalue 5 from EU on     *)
	(********************************************************************************************)
	(********************************************************************************************)

	(********************************************************************************************)
	(****************************** Q - L I M I T I N G *****************************************)
	(********************************************************************************************)
	(* Q - LIMITING 																			*)
	(*																							*)
	(*(DE)Activating  - HW --> To connection or to set fix value    		         		   	*)
	OUT_CU.bQLim_GenC_SetEUCOn	:= IN_CU.tQLim_GenC_SetEUCOn.Di;		(* DI: setpoint reactive power limitation (QLim) from EU - on (activate)   *)
	OUT_CU.bQLim_GenC_SetEUCOf	:= IN_CU.tQLim_GenC_SetEUCOf.Di;		(* DI: setpoint reactive power limitation (QLim) from EU - off (deactivate)*)

	(*(DE)Activating - BUS																		*)
	OUT_CU.bGenC_QLimBC_SetCOn; 				(* bus: setpoint reactive power limitation (QLim) from EU - on (activate)    *)
	OUT_CU.bGenC_QLimBC_SetCOf;			 		(* bus: setpoint reactive power limitation (QLim) from EU - off (deactivate) *)
	(*
	(* BUSSIGANAL connect  - Q Limiting EU          											*)
	(* to do:																					*)
	(* - BusSetpoint OUT_CU.rGenC_QLimBC              				 		                    *)
	(*  - OUT_CU.bGenC_QLimSetErrBC generieren - falls TRUE wird der Backupwert (Parameter) verwendet	 *)
	OUT_CU.rGenC_QLimBC;    	(* bus: scaling value for reactive power limitation for EVA BUS[kVAr]    *)
	OUT_CU.bGenC_QLimSetErrBC;	(* bus: setpoint reactive power limitation from EU error - use backupvalue*)

	(*- - - - - - - - - - - - - - - - -  F E E D B A C K  S I G N A L S  - - - - - - - - - - -  *)
	(* use the following variables as DO in the I/O configuration if needed 					*)
	(* QLim_GenC_SOn; (*  reactive power limiting (QLim)  is on                     			*)
	(* QLim_GenC_SOf; (*  reactive power limiting (QLim)  is off	                    		*)
	(* QLim_GenC_Act; (*  reactive power limiting (Plim) from EU is aktiv            			*)
	(********************************************************************************************)

	(********************************************************************************************)
	(*********************************** COS (PHI) - f(P) ***************************************)
	(********************************************************************************************)
	(*(DE)Activating  - HW --> To connect or to set fix value    		         				*)
	OUT_CU.bQPC_GenC_SetEUCOn	:= IN_CU.tQPC_GenC_SetEUCOn.Di;  			(*DI: setpoint reactive power characteristics COS(phi)=f(P) from EU - on (activate)    *)
	OUT_CU.bQPC_GenC_SetEUCOf	:= IN_CU.tQPC_GenC_SetEUCOf.Di := TRUE;  	(*DI: setpoint reactive power characteristics COS(phi)=f(P) from EU - off (deactivate) *)
	(*																							*)
	(*(DE)Activating - bus																		*)
	OUT_CU.bGenC_QPCBC_SetCOn; 				(* bus: setpoint reactive power characteristics COS(phi)=f(P) from EU - on (activate)	*)
	OUT_CU.bGenC_QPCBC_SetCOf	:= TRUE; 	(* bus: setpoint reactive power characteristics COS(phi)=f(P) from - off (deactivate)	*)
	(********************************************************************************************)

	(*- - - - - - - - - - - - - - - - -  F E E D B A C K  S I G N A L S  - - - - - - - - - - -  *)
	IN_CU.tQPC_GenC_SOn.Do; (*  reactive power characteristics COS(phi)=f(P) from EU is on		*)
	IN_CU.tQPC_GenC_SOf.Do; (*  reactive power characteristics COS(phi)=f(P) from EU is on		*)

	(********************************************************************************************)
	(********************************* U - S E T   V A L U E ************************************)
	(********************************************************************************************)
	(*																							*)
	OUT_CU.bUist_max 			:= FALSE;	(* TRUE = Uist für Q(U) & cosphi(U) ist max. Generatorspannung    *)
	(* Ph-Ph, FALSE = durchschnittliche Generatorspannung Ph-Ph 								*)
	(* Activation U setpoint for PF(U), Q(U) functions											*)
	OUT_CU.bGenC_UQBC_SetCOn;(* bus: setpoint generator voltage for rective power - on (activate)    *)
	OUT_CU.bGenC_UQBC_SetCOf	:= TRUE;	(* bus: setpoint generator voltage FOR rective power - off (deactivate)*)
	(* Activation U setpoint for U control														*)
	(*(DE)Activating  - HW --> To connect or to set fix value    		         				*)
	OUT_CU.bU_GenC_SetEUCOn; (*DI: setpoint generator voltage FOR voltage control - on (activate)    *)
	OUT_CU.bU_GenC_SetEUCOf := TRUE; (*DI: setpoint generator voltage FOR voltage control - off (deactivate)    *)
	(*																							*)
	(*(DE)Activating - bus																		*)
	OUT_CU.bGenC_UBC_SetCOn; (*bus: setpoint generator voltage FOR voltage control - on (activate)    *)
	OUT_CU.bGenC_UBC_SetCOf := TRUE; (*bus: setpoint generator voltage FOR voltage control - off (deactivate)
	(*																						    *)
	(* BUSSIGANAL connect  - Q Limiting EU          											*)
	(* to do:																		        	*)
	(* - BusSetpoint OUT_CU.rGenC_UQBC              				 		                    *)
	(* - OUT_CU.bU_GenC_SetErrBC generieren - falls TRUE wird der Backupwert (Parameter) verwendet	 		*)
	OUT_CU.rGenC_UQBC;    		(* bus: scaling value generator voltage for reactive power (Q) [1.00] = 100% from Nominal Value for Setpoint (Parameter 11696) *)
	OUT_CU.bU_GenC_SetErrBC;	(* bus: setpoint voltage from EU error - use backupvalue		*)

	(********************************************************************************************)
	(***************************************** Q(U) *********************************************)
	(********************************************************************************************)
	(*(DE)Activating  - HW --> To bind or to set fix value    		         					*)
	OUT_CU.bQUC_GenC_SetEUCOn	:= IN_CU.tQUC_GenC_SetEUCOn.Di;			(* DI: setpoint reactive power characteristics Q=f(U) from EU -on (activate)   *)
	OUT_CU.bQUC_GenC_SetEUCOf	:= IN_CU.tQUC_GenC_SetEUCOf.Di := TRUE;	(* DI: setpoint reactive power characteristics Q=f(U) from EU -off (deactivate)*)
	(*																							*)
	(*(DE)Activating - bus																		*)
	OUT_CU.bGenC_QUCBC_SetCOn; 				(* bus: setpoint reactive power characteristics Q=f(U) from EU -on (activate)   *)
	OUT_CU.bGenC_QUCBC_SetCOf	:= TRUE;	(* bus: setpoint reactive power characteristics Q=f(U) from EU -off (deactivate)*)
	(********************************************************************************************)

	(*- - - - - - - - - - - - - - - - -  F E E D B A C K  S I G N A L S  - - - - - - - - - - -  *)
	IN_CU.tQUC_GenC_SOn.Do;     (*  reactive power characteristics Q=f(U) from EU is on       	*)
	IN_CU.tQUC_GenC_SOf.Do;     (*  reactive power characteristics Q=f(U) from EU is off       	*)
	(********************************************************************************************)

	(********************************************************************************************)
	(*********************************** COS (PHI) - f(U) ***************************************)
	(********************************************************************************************)
	(*(DE)Activating  - HW --> To bind or to set fix value    		         					*)
	OUT_CU.bPFUC_GenC_SetEUCOn	:= IN_CU.tPFUC_GenC_SetEUCOn.Di; 		(* DI: setpoint reactive power characteristics COS(phi)=f(U) von EU -on (active)    		 *)
	OUT_CU.bPFUC_GenC_SetEUCOf	:= IN_CU.tPFUC_GenC_SetEUCOf.Di:=TRUE; 	(* DI: setpoint reactive power characteristics COS(phi)=f(U) von EU -off (deactive) *)
	(*																							*)
	(*(DE)Activating - bus																		*)
	OUT_CU.bGenC_PFUCBC_SetCOn;					 (* bus: setpoint reactive power characteristics COS(phi)=f(U) from EU -on (active)   *)
	OUT_CU.bGenC_PFUCBC_SetCOf	:= TRUE;		 (* bus: setpoint reactive power characteristics COS(phi)=f(U) from EU -off (deactive)*)

	(*- - - - - - - - - - - - - - - - -  F E E D B A C K  S I G N A L S  - - - - - - - - - - -  *)
	IN_CU.tPFUC_GenC_SOn.Do;	   (*  reactive power characteristics COS(phi)=f(P) from EU is on  *)
	IN_CU.tPFUC_GenC_SOf.Do;       (*  reactive power characteristics COS(phi)=f(P) from EU is off *)
	(********************************************************************************************)

	(********************************************************************************************)
	(*********************************** Q - f(P) ***********************************************)
	(********************************************************************************************)
	(*(DE)Activating  - HW --> To bind or to set fix value    		         					*)
	OUT_CU.bQP_GenC_SetEUCOn := IN_CU.tQP_GenC_SetEUCOn.Di; 		(* DI: setpoint reactive power characteristics Q=f(P) von EU -on (active)    		 *)
	OUT_CU.bQP_GenC_SetEUCOf := IN_CU.tQP_GenC_SetEUCOf.Di:= TRUE; 	(* DI: setpoint reactive power characteristics Q=f(P) von EU -off (deactive) *)
	(*																							*)
	(*(DE)Activating - bus																		*)
	OUT_CU.bGenC_QPBC_SetCOn;			 (* bus: setpoint reactive power characteristics Q=f(P) from EU -on (active)   *)
	OUT_CU.bGenC_QPBC_SetCOf	:= TRUE; (* bus: setpoint reactive power characteristics Q=f(P) from EU -off (deactive)*)

	(*- - - - - - - - - - - - - - - - -  F E E D B A C K  S I G N A L S  - - - - - - - - - - -  *)
	IN_CU.tQP_GenC_SOn.Do;	   (*  reactive power characteristics Q=f(P) from EU is on  *)
	IN_CU.tQP_GenC_SOf.Do;       (*  reactive power characteristics Q=f(P) from EU is off *)
	(********************************************************************************************)

	(********************************************************************************************)
	(*************** P R I O R I T I Z A T I O N  T H E  F U N C T I O N S **********************)
	(********************************************************************************************)
	(* Prioritization the EU Functions for voltage controling									*)
	(* the smaller number the greater priority													*)
	(* SEVERAL FUNCTIONS AT THE SAME TIME SPORTS - "WINNING" THE ONE WITH PRIORITY           	*)
	OUT_CU.iGenC_PrioQCustSet := 9;		(* Prioritet  reactive power Q customized						*)
	OUT_CU.iGenC_PrioQUset   := 7;		(* Prioritet  reactive power U control(Q) -                     *)
	OUT_CU.iGenC_PrioQ   	 := 6;		(* Prioritet  reactive power (Q) - fixvalue                     *)
	OUT_CU.iGenC_PrioQP		 := 5;		(* Prioritet  reactive power characteristic Q=f(P)              *)
	OUT_CU.iGenC_PrioQUC     := 4;		(* Prioritet  reactive power characteristic Q=f(U)              *)
	OUT_CU.iGenC_PrioPFUC    := 3;		(* Prioritet  reactive power characteristic COS(phi)=f(U)       *)
	OUT_CU.iGenC_PrioPFPC    := 2;		(* Prioritet  reactive power characteristic COS(phi)=f(P)       *)
	OUT_CU.iGenC_PrioPF      := 1;		(* Prioritet  genetaror power factor (COS(phi)) - fixvalue      *)
	(********************************************************************************************)

	(********************************************************************************************)
	(*************** POINT OF REFERENCE (POR) - CUSTOMIZED **************************************)
	(********************************************************************************************)
	(* To do if customized point of reference is selected   									*)
	(* Para.iQ_GrC_PointRef = 0																	*)
	(* - provide actual active power  OUT_CU.rP_POR_Act_Cust								        *)
	(* - provide actual voltage OUT_CU.rU_POR_Act_Cust		     		      				        *)

	OUT_CU.rP_POR_Act_Cust; (* actual active power used as point of reference [kW] - connect spare AI e.g IN_CU.tCustAnaIn[1].Ai*)
	OUT_CU.rU_POR_Act_Cust;	(* actual voltage used as point of reference [V] - connect spare AI e.g IN_CU.tCustAnaIn[1].Ai*)
	(********************************************************************************************)

	(********************************************************************************************)
	(*************** POINT OF CONTROL (POC)- CUSTOMIZED ********************************************)
	(********************************************************************************************)
	(* To do if customized point of control is selected   										*)
	(* Para.iQ_GrC_PointCtrl = 0																*)
	(*(AI)Activating  - HW --> To connect spare AI                      		         		*)
	OUT_CU.rS_POC_Act_Cust;(*  := IN_CU.tCustAnaIn[1].Ai; (* AI: apparent power custom measurement [kVA] *)
	OUT_CU.rP_POC_Act_Cust;(*  := IN_CU.tCustAnaIn[2].Ai; (* AI: active   power custom measurement [kW]	 *)
	OUT_CU.rQ_POC_Act_Cust;(*  := IN_CU.tCustAnaIn[3].Ai; (* AI: reactive power custom measurement [kVAr]*)
	OUT_CU.rPF_POC_Act_Cust;(* := IN_CU.tCustAnaIn[4].Ai; (* AI: power factor   custom measurement       *)

	(*rS_POC_Act_Cust calculation if value is not available - - - - - - - - - - - - - - - - - - - - *)(*
	OUT_CU.rS_POC_Act_Cust  := SQRT(OUT_CU.rP_POC_Act_Cust * OUT_CU.rP_POC_Act_Cust + OUT_CU.rQ_POC_Act_Cust * OUT_CU.rQ_POC_Act_Cust);

	(*rPF_POC_Act_Cust calculation if value is not available - - - - - - - - - - - - - - - - - - - - *)(*
	IF OUT_CU.rS_POC_Act_Cust > 0 THEN
		OUT_CU.rPF_POC_Act := OUT_CU.rP_POC_Act_Cust / OUT_CU.rS_POC_Act_Cust;
	END_IF;
	(********************************************************************************************)

	(********************************************************************************************)
	(*************** Q FUNCTION #0 - CUSTOMIZED  ************************************************)
	(********************************************************************************************)
	(* (DE)activation - bus          		         					        	            *)
	OUT_CU.bGenC_QCustBC_SetCOn;			(*bus: Customized Q setpoint		 - on (activate)*)
	OUT_CU.bGenC_QCustBC_SetCOf	:= TRUE;	(*bus: Customized Q setpoint	  - off (deactivate)*)

	(* to do:																		        	*)
	(* - Q setpoint	 OUT_CU.rQ_Cust		              				 		                    *)
	OUT_CU.rQ_Cust;				(* Customized Q setpoint [kVAr]- connect spare AI e.g IN_CU.tCustAnaIn[1].Ai*)
	(********************************************************************************************)

	(********************************************************************************************)
	(********************************************************************************************)
	(*************** W I R K L E I S T U N G ** / ** A C T I V E   P O W E R ********************)
	(********************************************************************************************)
	(********************************************************************************************)

	(********************************************************************************************)
	(*************************** P - S E T   V A L U E ******************************************)
	(********************************************************************************************)
	(*(DE)Activating  - HW --> To connect or to set fix value    		         		  	    *)
	OUT_CU.bP_GenC_SetEUCOn := IN_CU.tP_GenC_SetEUCOn.Di;  (* DI: request power value from EU - on (activate)	        *)
	OUT_CU.bP_GenC_SetEUCOf := IN_CU.tP_GenC_SetEUCOf.Di:=TRUE;	(* DI: request power value from EU - off (deactivate)   *)

	(*Digitalinputs for power fixvalue - in I/O list bind if needed	                			*)
	OUT_CU.P_GenC_SetFix1 := IN_CU.tP_GenC_SetFix1EU.Di; (* DI: power value - P- fixvalue 1 from EU  *)
	OUT_CU.P_GenC_SetFix2 := IN_CU.tP_GenC_SetFix2EU.Di; (* DI: power value - P- fixvalue 2 from EU  *)
	OUT_CU.P_GenC_SetFix3 := IN_CU.tP_GenC_SetFix3EU.Di; (* DI: power value - P- fixvalue 3 from EU  *)
	OUT_CU.P_GenC_SetFix4 := IN_CU.tP_GenC_SetFix4EU.Di; (* DI: power value - P- fixvalue 4 from EU  *)
	OUT_CU.P_GenC_SetFix5 := IN_CU.tP_GenC_SetFix5EU.Di; (* DI: power value - P- fixvalue 5 from EU  *)
	(*																							*)
	(*(DE)Activating - bus																		*)
	OUT_CU.bGenC_PBC_SetCOn; 			(* bus: setpoint power P from EU -on (activate) 	    *)
	OUT_CU.bGenC_PBC_SetCOf	:= TRUE; 	(* bus: setpoint power P from EU -off (deactivate) 		*)
	(*
	(* BUSSIGNAL connection  - P Set value from EU         										*)
	(* to do:																		        	*)
	(* - BusSetpoint OUT_CU.rGenC_PBC	              				 		                    *)
	(* - OUT_CU.bP_GenC_SetErr generieren - falls TRUE wird der Backupwert (Parameter) verwendet*)
	OUT_CU.rGenC_PBC;        (* bus: scaling value for power P from EU 	[kW]					*)
	OUT_CU.bP_GenC_SetErr;   (* Generator power setpoint measuring signal failure 				*)

	(*- - - - - - - - - - - - - - - - -  F E E D B A C K  S I G N A L S  - - - - - - - - - - -  *)
	IN_CU.tP_GenC_SOn.Do; (*  power value fon EU is on  	 *)
	IN_CU.tP_GenC_SOf.Do; (*  power value fon EU is off      *)
	(********************************************************************************************)

	(********************************************************************************************)
	(****************************** P - L I M I T I N G *****************************************)
	(********************************************************************************************)
	(*(DE)Activating  - HW --> To connect or to set fix value    		         				*)
	IF NOT Para.bDEIE_Active THEN
		OUT_CU.bPLim_GenC_SetEUCOn := IN_CU.tPLim_GenC_SetEUCOn.Di := TRUE; (* DI: setpoint power limitation (Plim) from EU - on (activate)    	*)
		OUT_CU.bPLim_GenC_SetEUCOf := IN_CU.tPLim_GenC_SetEUCOf.Di := TRUE; (* DI: setpoint power limitation (Plim) from EU - off (deactivate) 	*)
	ELSE
		OUT_CU.bPLim_GenC_SetEUCOn := IN_CU.tPLim_GenC_SetEUCOn.Di;(*<-- DON'T change - just for ERDF / DEIE*)
		OUT_CU.bPLim_GenC_SetEUCOf := IN_CU.tPLim_GenC_SetEUCOf.Di;(*<-- DON'T change - just for ERDF / DEIE*)
	END_IF;
	(*																							*)
	(* Marshalling DI: P - Limiting/reduction fixed value for singel-steps		     		    *)
	OUT_CU.PLim_GenC_SetEUPFix1 := IN_CU.tPLim_GenC_SetEUPFix1.Di;(* DI: power limitation fixvalue 1 *)
	OUT_CU.PLim_GenC_SetEUPFix2 := IN_CU.tPLim_GenC_SetEUPFix2.Di;(* DI: power limitation fixvalue 2 *)
	OUT_CU.PLim_GenC_SetEUPFix3 := IN_CU.tPLim_GenC_SetEUPFix3.Di;(* DI: power limitation fixvalue 2 *)
	OUT_CU.PLim_GenC_SetEUPFix4 := IN_CU.tPLim_GenC_SetEUPFix4.Di;(* DI: power limitation fixvalue 3 *)
	OUT_CU.PLim_GenC_SetEUPFix5 := IN_CU.tPLim_GenC_SetEUPFix5.Di;(* DI: power limitation fixvalue 5 *)
	(*(DE)Activating - bus																	   	*)
	OUT_CU.bGenC_PLimBC_SetCOn;				(* bus: power limition from  EU - on (activate)     *)
	OUT_CU.bGenC_PLimBC_SetCOf	:= TRUE;	(* bus: power limition from  EU - off (deactivate)  *)

	(* BUSSIGANAL connect - power limiting EU                                                   *)
	(* to do:																		          	*)
	(* - BusSetpoint OUT_CU.rGenC_PLimBC	              				 		                *)
	(* - OUT_CU.bP_GenC_SetErrPlim generieren - falls TRUE wird der Backupwert (Parameter) verwendet *)
	OUT_CU.rGenC_PLimBC;		(* bus: scaling value power limitation from EU [kW]           	*)
	OUT_CU.bP_GenC_SetErrPlim;	(* power limitation BUS EU error - use backupvalue			    *)

	(*- - - - - - - - - - - - -  F E E D B A C K  S I G N A L S  - - - - - - - - - - - - - - -  *)
	IN_CU.tPLim_GenC_SOn.Do;  (*  power limitation (PLim) from EU is on							*)
	IN_CU.tPLim_GenC_SOf.Do;  (*  power limitation (Plim) from EU is off						*)
	IN_CU.tPLim_GenC_Act.Do;  (*  power limitation (Plim) from EU is aktiv						*)
	IN_CU.tP_GenC_Fix0SOn.Do; (*  no limiting power value - P- fixvalue 0 from EU is on			*)
	IN_CU.tP_GenC_Fix1SOn.Do; (*  power value - P- fixvalue 1 from EU is on						*)
	IN_CU.tP_GenC_Fix2SOn.Do; (*  power value - P- fixvalue 2 from EU is on						*)
	IN_CU.tP_GenC_Fix3SOn.Do; (*  power value - P- fixvalue 3 from EU is on						*)
	IN_CU.tP_GenC_Fix4SOn.Do; (*  power value - P- fixvalue 4 from EU is on						*)
	IN_CU.tP_GenC_Fix5SOn.Do; (*  power value - P- fixvalue 5 from EU is on						*)
	IN_CU.tEU_RM_BLOCK.Do;	  (*  Separate unit of utility and of active network              	*)
	(********************************************************************************************)

	(********************************************************************************************)
	(************** PFC - P r i m a r y F r e q u e n c y C o n t r o l *************************)
	(********************************************************************************************)
	(*(DE)Activating  - HW --> To connect or to set fix value    		         			    *)
	OUT_CU.bPFC_SetCOn	:= IN_CU.tPFC_SetCOn.Di; 		(* DI:primary frequency control - on (activate)	*)
	OUT_CU.bPFC_SetCOf	:= IN_CU.tPFC_SetCOf.Di :=TRUE; (* DI:primary frequency control - off (deactivate)	*)
	(*																							*)
	(*(DE)Activating - bus																		*)
	OUT_CU.bGenC_PFCBC_SetCOn; 				(* bus: primary frequency control - on (activate)	*)
	OUT_CU.bGenC_PFCBC_SetCOf	:= TRUE; 	(* bus: primary frequency control - off (deactivate)*)

	(*- - - - - - - - - - - F E E D B A C K  S I G N A L S  - - - - - - - - - - - - - -- - - -  *)
	IN_CU.tPFC_SOn.Do;		(*  primary frequency control is on									*)
	IN_CU.tPFC_SOf.Do;    	(*  primary frequency control is off								*)
	(********************************************************************************************)

	(********************************************************************************************)
	(************** RMC - R e g u l a t i n g M a r g i n C o n t r o l *************************)
	(********************************************************************************************)
	(*(DE)Activating  - HW --> To connect or to set fix value    		         			    *)
	OUT_CU.bRMC_SetCOn	:= IN_CU.tRMC_SetCOn.Di; (* DI:regulation margin control -on (activate)	*)
	OUT_CU.bRMC_SetCOf	:= IN_CU.tRMC_SetCOf.Di :=TRUE; (* DI:regulation margin control -off (deactivate) *)
	(*																							*)
	(*(DE)Activating - bus																		*)
	OUT_CU.bGenC_RMCBC_SetCOn; 				(* bus: regulation margin control -on (activate)	*)
	OUT_CU.bGenC_RMCBC_SetCOf	:= TRUE; 	(* bus: regulation margin control -off (deactivate)	*)

	(*- - - - - - - - - - - F E E D B A C K  S I G N A L S  - - - - - - - - - - - - - -- - - -  *)
	IN_CU.tRMC_SOn.Do; 		(*  regulation margin control is on									*)
	IN_CU.tRMC_SOf.Do;		(*  regulation margin control is off								*)
	(********************************************************************************************)

	(********************************************************************************************)
	(************************** E R D F *********************************************************)
	(********************************************************************************************)
	(* Enable the functionality for the ERDF customers now via Parameter *)
	(* electrical / grid / static grid code *)
	(********************************************************************************************)

	(********************************************************************************************)
	(************** FSM - F r e q u e n c y C o n t r o l *************************)
	(********************************************************************************************)
	(*(DE)Activating  - HW --> To connect or to set fix value    		         			    *)
	OUT_CU.bFC_SetCOn	:= IN_CU.tSet_FC_COn.Di; 		(* DI: frequency control - on (activate)	*)
	OUT_CU.bFC_SetCOf	:= IN_CU.tSet_FC_COf.Di :=TRUE; (* DI: frequency control - off (deactivate)	*)
	(*																							*)
	(*(DE)Activating - bus																		*)
	OUT_CU.bSet_FC_COn_Bus; 				(* bus: primary frequency control - on (activate)	*)
	OUT_CU.bSet_FC_COf_Bus	:= TRUE; 		(* bus: primary frequency control - off (deactivate)*)

	(*- - - - - - - - - - - F E E D B A C K  S I G N A L S  - - - - - - - - - - - - - -- - - -  *)
	IN_CU.tFC_SOn.Do;		(*  primary frequency control is on								*)
	IN_CU.tFC_SOf.Do;    	(*  primary frequency control is off								*)
	(********************************************************************************************)

	(********************************************************************************************)
	(************************* P(U) - ÖSTERREICH*************************************************)
	(********************************************************************************************)
	(*(DE)Activating  - HW --> To connect or to set fix value    		         			    *)
	OUT_CU.bPU_SetCOn	:= IN_CU.tSet_PU_COn.Di; 		(* DI: frequency control - on (activate)	*)
	OUT_CU.bPU_SetCOf	:= IN_CU.tSet_PU_COf.Di :=TRUE; (* DI: frequency control - off (deactivate)	*)
	(*																							*)
	(*(DE)Activating - bus																		*)
	OUT_CU.bGenC_PUBC_SetCOn; 				(* bus: P(U) - Österreich - on (activate)	*)
	OUT_CU.bGenC_PUBC_SetCOf := TRUE; 		(* bus: P(U) - Österreich - off (deactivate)*)

	(*- - - - - - - - - - - F E E D B A C K  S I G N A L S  - - - - - - - - - - - - - -- - - -  *)
	IN_CU.tPU_SOn.Do;		(*  P(U) Österreich is on								*)
	IN_CU.tPU_SOn.Do;    	(*  P(U) Österreich is off								*)
	(********************************************************************************************)

	(********************************************************************************************)
	(************************* Parameter External************************************************)
	(********************************************************************************************)
	(************************* Frequency Deadband LFSMO******************************************)
	(*Activating - HW --> To connect or to set fix value    		         			   		*)
	OUT_CU.tCU2GR.bLFSMO_DB_AI_COn := IN_CU.tHA2CU.tSet_LFSMO_DB_COn.Di;
	OUT_CU.tCU2GR.bLFSMO_DB_AI_COf := IN_CU.tHA2CU.tSet_LFSMO_DB_COf.Di := TRUE;
	(*
	(*Activating - via Bus signal																*)
	OUT_CU.tCU2GR.bLFSMO_DB_BC_COn;
	OUT_CU.tCU2GR.bLFSMO_DB_BC_COf := TRUE;
	(*																							*)
	(* BUSSIGNAL connection  - Frequency Limit LFSMO from EU            						*)
	(* to do:																		        	*)
	(* - BusSetpoint OUT_CU.tCU2GR.rF_LFSMO_DB_BC      				 		                    *)
	(* - OUT_CU.tCU2GR.bLFSMO_DB_BC_SetErr - falls TRUE wird der Backupwert (Parameter) verwendet  *)
	OUT_CU.tCU2GR.rF_LFSMO_DB_BC;        (* bus: scaling value for Frequency Deadband LFSMO from EU [Hz] *)
	OUT_CU.tCU2GR.bLFSMO_DB_BC_SetErr;   (* Frequency Limit LFSMO measuring signal failure   	*)
	(********************************************************************************************)
	(************************* Frequency Deadband LFSMU******************************************)
	(*Activating - HW --> To connect or to set fix value    		         			   		*)
	OUT_CU.tCU2GR.bLFSMU_DB_AI_COn := IN_CU.tHA2CU.tSet_LFSMU_DB_COn.Di;
	OUT_CU.tCU2GR.bLFSMU_DB_AI_COf := IN_CU.tHA2CU.tSet_LFSMU_DB_COf.Di := TRUE;
	(*
	(*Activating - via Bus signal																*)
	OUT_CU.tCU2GR.bLFSMU_DB_BC_COn;
	OUT_CU.tCU2GR.bLFSMU_DB_BC_COf := TRUE;
	(*																							*)
	(* BUSSIGNAL connection  - Frequency Limit LFSMU from EU            						*)
	(* to do:																		        	*)
	(* - BusSetpoint OUT_CU.tCU2GR.rF_LFSMU_DB_BC      				 		                    *)
	(* - OUT_CU.tCU2GR.bLFSMU_DB_BC_SetErr generieren - falls TRUE wird der Backupwert (Parameter) verwendet*)
	OUT_CU.tCU2GR.rF_LFSMU_DB_BC;        (* bus: scaling value for Frequency Limit LFSMU from EU [Hz] *)
	OUT_CU.tCU2GR.bLFSMU_DB_BC_SetErr;   (* Frequency Limit LFSMU measuring signal failure  	*)
	(********************************************************************************************)
	(************************* Positive Droop LFSMO**********************************************)
	(*Activating - HW --> To connect or to set fix value    		         			   		*)
	OUT_CU.tCU2GR.bLFSMO_Droop_AI_COn := IN_CU.tHA2CU.tSet_LFSMO_Droop_COn.Di;
	OUT_CU.tCU2GR.bLFSMO_Droop_AI_COf := IN_CU.tHA2CU.tSet_LFSMO_Droop_COf.Di := TRUE;
	(*
	(*Activating - via Bus signal																*)
	OUT_CU.tCU2GR.bLFSMO_Droop_BC_COn;
	OUT_CU.tCU2GR.bLFSMO_Droop_BC_COf := TRUE;
	(*																							*)
	(* BUSSIGNAL connection  - Positive Droop LFSMO from EU             						*)
	(* to do:																		        	*)
	(* - BusSetpoint OUT_CU.tCU2GR.rP_LFSMO_Droop_BC	              				 		                    *)
	(* - OUT_CU.tCU2GR.bLFSMO_Droop_BC_SetErr generieren - falls TRUE wird der Backupwert (Parameter) verwendet*)
	OUT_CU.tCU2GR.rP_LFSMO_Droop_BC;        (* bus: scaling value for Positive Droop LFSMO from EU [%] *)
	OUT_CU.tCU2GR.bLFSMO_Droop_BC_SetErr;   (* Positive Droop LFSMO measuring signal failure	*)
	(********************************************************************************************)
	(************************* Negative Droop LFSMU**********************************************)
	(*Activating - HW --> To connect or to set fix value    		         			   		*)
	OUT_CU.tCU2GR.bLFSMU_Droop_AI_COn := IN_CU.tHA2CU.tSet_LFSMU_Droop_COn.Di;
	OUT_CU.tCU2GR.bLFSMU_Droop_AI_COf := IN_CU.tHA2CU.tSet_LFSMU_Droop_COf.Di := TRUE;
	(*
	(*Activating - via Bus signal																*)
	OUT_CU.tCU2GR.bLFSMU_Droop_BC_COn;
	OUT_CU.tCU2GR.bLFSMU_Droop_BC_COf := TRUE;
	(*																							*)
	(* BUSSIGNAL connection  - Negative droop LFSMU from EU         		    				*)
	(* to do:																		        	*)
	(* - BusSetpoint OUT_CU.tCU2GR.rP_LFSMU_Droop_BC   				 		                    *)
	(* - OUT_CU.tCU2GR.bLFSMU_Droop_BC_SetErr generieren - falls TRUE wird der Backupwert (Parameter) verwendet*)
	OUT_CU.tCU2GR.rP_LFSMU_Droop_BC;        (* bus: scaling value for Negative Droop LFSMU from EU [%] *)
	OUT_CU.tCU2GR.bLFSMU_Droop_BC_SetErr;   (* Negative Droop LFSMU measuring signal failure    *)
	(********************************************************************************************)
	(************************* Droop FSMU********************************************************)
	(*Activating - HW --> To connect or to set fix value    		         			   		*)
	OUT_CU.tCU2GR.bFSMU_Droop_AI_COn := IN_CU.tHA2CU.tSet_FSMU_Droop_COn.Di;
	OUT_CU.tCU2GR.bFSMU_Droop_AI_COf := IN_CU.tHA2CU.tSet_FSMU_Droop_COf.Di := TRUE;
	(*
	(*Activating - via Bus signal																*)
	OUT_CU.tCU2GR.bFSMU_Droop_BC_COn;
	OUT_CU.tCU2GR.bFSMU_Droop_BC_COf := TRUE;
	(*																							*)
	(* BUSSIGNAL connection  - Droop FSMU from EU				         						*)
	(* to do:																		        	*)
	(* - BusSetpoint OUT_CU.tCU2GR.rP_FSMU_Droop_BC	              				 		        *)
	(* - OUT_CU.tCU2GR.bFSMU_Droop_BC_SetErr generieren - falls TRUE wird der Backupwert (Parameter) verwendet*)
	OUT_CU.tCU2GR.rP_FSMU_Droop_BC;        (* bus: scaling value for Droop FSMU from EU	[%]		*)
	OUT_CU.tCU2GR.bFSMU_Droop_BC_SetErr;   (* Droop FSMU measuring signal failure	            *)
	(********************************************************************************************)
	(************************* Droop FSMO********************************************************)
	(*Activating - HW --> To connect or to set fix value    		         			   		*)
	OUT_CU.tCU2GR.bFSMO_Droop_AI_COn := IN_CU.tHA2CU.tSet_FSMO_Droop_COn.Di;
	OUT_CU.tCU2GR.bFSMO_Droop_AI_COf := IN_CU.tHA2CU.tSet_FSMO_Droop_COf.Di := TRUE;
	(*
	(*Activating - via Bus signal																*)
	OUT_CU.tCU2GR.bFSMO_Droop_BC_COn;
	OUT_CU.tCU2GR.bFSMO_Droop_BC_COf := TRUE;
	(*																							*)
	(* BUSSIGNAL connection  - Droop FSMO from EU                       						*)
	(* to do:																		        	*)
	(* - BusSetpoint OUT_CU.tCU2GR.rP_FSMO_Droop_BC    				 		                    *)
	(* - OUT_CU.tCU2GR.bFSMO_Droop_BC_SetErr generieren - falls TRUE wird der Backupwert (Parameter) verwendet*)
	OUT_CU.tCU2GR.rP_FSMO_Droop_BC;        (* bus: scaling value for Droop FSMO from EU [%]  	*)
	OUT_CU.tCU2GR.bFSMO_Droop_BC_SetErr;   (* Droop FSMO measuring signal failure               *)
	(********************************************************************************************)
	(************************* Deadband FSMU*****************************************************)
	(*Activating - HW --> To connect or to set fix value    		         			   		*)
	OUT_CU.tCU2GR.bFSMU_DB_AI_COn := IN_CU.tHA2CU.tSet_FSMU_DB_COn.Di;
	OUT_CU.tCU2GR.bFSMU_DB_AI_COf := IN_CU.tHA2CU.tSet_FSMU_DB_COf.Di := TRUE;
	(*
	(*Activating - via Bus signal																*)
	OUT_CU.tCU2GR.bFSMU_DB_BC_COn;
	OUT_CU.tCU2GR.bFSMU_DB_BC_COf := TRUE;
	(*																							*)
	(* BUSSIGNAL connection  -Deadband FSMU from EU				         						*)
	(* to do:																		        	*)
	(* - OUT_CU.tCU2GR.rF_FSMU_DB_BC	              				 		                    *)
	(* - OUT_CU.tCU2GR.bFSMU_DB_BC_SetErr generieren - falls TRUE wird der Backupwert (Parameter) verwendet*)
	OUT_CU.tCU2GR.rF_FSMU_DB_BC;           (* bus: scaling value for Deadband FSMU from EU [Hz] *)
	OUT_CU.tCU2GR.bFSMU_DB_BC_SetErr;      (* Deadband FSMU measuring signal failure	    	*)
	(********************************************************************************************)
	(************************* Deadband FSMO*****************************************************)
	(*Activating - HW --> To connect or to set fix value    		         			   		*)
	OUT_CU.tCU2GR.bFSMO_DB_AI_COn := IN_CU.tHA2CU.tSet_FSMO_DB_COn.Di;
	OUT_CU.tCU2GR.bFSMO_DB_AI_COf := IN_CU.tHA2CU.tSet_FSMO_DB_COf.Di := TRUE;
	(*
	(*Activating - via Bus signal																*)
	OUT_CU.tCU2GR.bFSMO_DB_BC_COn;
	OUT_CU.tCU2GR.bFSMO_DB_BC_COf := TRUE;
	(*																							*)
	(* BUSSIGNAL connection  - Deadband FSMO from EU         			            			*)
	(* to do:																		        	*)
	(* - BusSetpoint OUT_CU.tCU2GR.rF_FSMO_DB_BC       				 		                    *)
	(* - OUT_CU.tCU2GR.bFSMO_DB_BC_SetErr - falls TRUE wird der Backupwert (Parameter) verwendet*)
	OUT_CU.tCU2GR.rF_FSMO_DB_BC;        (* bus: scaling value for Deadband FSMO from EU [Hz]    *)
	OUT_CU.tCU2GR.bFSMO_DB_BC_SetErr;  	(* Deadband FSMO measuring signal failure	            *)
	(********************************************************************************************)
	(************************* Positive Margin FSM***********************************************)
	(*Activating - HW --> To connect or to set fix value    		         			   		*)
	OUT_CU.tCU2GR.bFSM_RMC_Up_AI_COn := IN_CU.tHA2CU.tSet_FSM_RMC_Up_COn.Di;
	OUT_CU.tCU2GR.bFSM_RMC_Up_AI_COf := IN_CU.tHA2CU.tSet_FSM_RMC_Up_COf.Di := TRUE;
	(*
	(*Activating - via Bus signal																*)
	OUT_CU.tCU2GR.bFSM_RMC_Up_BC_COn;
	OUT_CU.tCU2GR.bFSM_RMC_Up_BC_COf := TRUE;
	(*																							*)
	(* BUSSIGNAL connection  - Positive Margin FSM from EU                 						*)
	(* to do:																		        	*)
	(* - BusSetpoint OUT_CU.tCU2GR.rP_FSM_RMC_Up_BC    				 		                    *)
	(* - OUT_CU.tCU2GR.bFSM_RMC_Up_BC_SetErr generieren - falls TRUE wird der Backupwert (Parameter) verwendet*)
	OUT_CU.tCU2GR.rP_FSM_RMC_Up_BC;       (* bus: scaling value for Positive Margin FSM from EU [%Pn] *)
	OUT_CU.tCU2GR.bFSM_RMC_Up_BC_SetErr;  (* Positive Margin FSM measuring signal failure       *)
	(********************************************************************************************)
	(************************* Negative Margin FSM***********************************************)
	(*Activating - HW --> To connect or to set fix value    		         			   		*)
	OUT_CU.tCU2GR.bFSM_RMC_Down_AI_COn := IN_CU.tHA2CU.tSet_FSM_RMC_Down_COn.Di;
	OUT_CU.tCU2GR.bFSM_RMC_Down_AI_COf := IN_CU.tHA2CU.tSet_FSM_RMC_Down_COf.Di := TRUE;
	(*
	(*Activating - via Bus signal																*)
	OUT_CU.tCU2GR.bFSM_RMC_Down_BC_COn;
	OUT_CU.tCU2GR.bFSM_RMC_Down_BC_COf := TRUE;
	(*																							*)
	(* BUSSIGNAL connection  - Negative Margin FSM from EU         					        	*)
	(* to do:																		        	*)
	(* - BusSetpoint OUT_CU.tCU2GR.rP_FSM_RMC_Down_BC  				 		                    *)
	(* - OUT_CU.tCU2GR.bFSM_RMC_Down_BC_SetErr generieren - falls TRUE wird der Backupwert (Parameter) verwendet*)
	OUT_CU.tCU2GR.rP_FSM_RMC_Down_BC;        (* bus: scaling value for Negative Margin FSM from EU [%Pn] *)
	OUT_CU.tCU2GR.bFSM_RMC_Down_BC_SetErr;   (* Negative Margin FSM measuring signal failure    *)
	(********************************************************************************************)
	(************************* Droop U***********************************************************)
	(*Activating - HW --> To connect or to set fix value    		         			   		*)
	OUT_CU.tCU2GR.bU_Droop_AI_COn := IN_CU.tHA2CU.tSet_U_Droop_COn.Di;
	OUT_CU.tCU2GR.bU_Droop_AI_COf := IN_CU.tHA2CU.tSet_U_Droop_COf.Di := TRUE;
	(*
	(*Activating - via Bus signal																*)
	OUT_CU.tCU2GR.bU_Droop_BC_COn;
	OUT_CU.tCU2GR.bU_Droop_BC_COf := TRUE;
	(*																							*)
	(* BUSSIGNAL connection  - Droop U from EU         					                    	*)
	(* to do:																		        	*)
	(* - BusSetpoint OUT_CU.tCU2GR.rU_Droop_BC         				 		                    *)
	(* - OUT_CU.tCU2GR.bU_Droop_BC_SetErr generieren - falls TRUE wird der Backupwert (Parameter) verwendet*)
	OUT_CU.tCU2GR.rU_Droop_BC;          (* bus: scaling value for Droop U from EU [%]           *)
	OUT_CU.tCU2GR.bU_Droop_BC_SetErr;   (* Droop U measuring signal failure                     *)
	(********************************************************************************************)
	(************************* Rampe rate********************************************************)
	(*Activating - HW --> To connect or to set fix value    		         			   		*)
	OUT_CU.tCU2GR.bFSM_Rmp_AI_COn := IN_CU.tHA2CU.tSet_FSM_Rmp_COn.Di;
	OUT_CU.tCU2GR.bFSM_Rmp_AI_COf := IN_CU.tHA2CU.tSet_FSM_Rmp_COf.Di := TRUE;
	(*
	(*Activating - via Bus signal																*)
	OUT_CU.tCU2GR.bFSM_Rmp_BC_COn;
	OUT_CU.tCU2GR.bFSM_Rmp_BC_COf := TRUE;
	(*																							*)
	(* BUSSIGNAL connection  - Rampe rate UP from EU         					            	*)
	(* to do:																		        	*)
	(* - BusSetpoint OUT_CU.tCU2GR.rP_FSM_Rmp_Up_BC and OUT_CU.tCU2GR.rP_FSM_Rmp_Down_BC        *)
	(* - OUT_CU.tCU2GR.bFSM_Rmp_BC_SetErr generieren - falls TRUE wird der Backupwert (Parameter) verwendet*)
	OUT_CU.tCU2GR.rP_FSM_Rmp_Up_BC;      (* bus: scaling value for Rampe rate UP from EU [%Pnom/s]	    *)
	OUT_CU.tCU2GR.rP_FSM_Rmp_Down_BC;    (* bus: scaling value for Rampe rate DOWN from EU [%Pnom/s]	    *)
	OUT_CU.tCU2GR.bFSM_Rmp_BC_SetErr;    (* Rampe rate measuring signal failure                 *)
	(********************************************************************************************)
	(************************* Reference Frequency FSM/LFSM**************************************)
	(*Activating - HW --> To connect or to set fix value    		         			   		*)
	OUT_CU.tCU2GR.bF_Ref_FSM_AI_COn := IN_CU.tHA2CU.tSet_F_Ref_FSM_COn.Di;
	OUT_CU.tCU2GR.bF_Ref_FSM_AI_COf := IN_CU.tHA2CU.tSet_F_Ref_FSM_COf.Di := TRUE;
	(*
	(*Activating - via Bus signal																*)
	OUT_CU.tCU2GR.bF_Ref_FSM_BC_COn;
	OUT_CU.tCU2GR.bF_Ref_FSM_BC_COf := TRUE;
	(*																							*)
	(* BUSSIGNAL connection  - Reference Frequency FSM/LFSM from EU         	            	*)
	(* to do:																		        	*)
	(* - BusSetpoint OUT_CU.tCU2GR.rF_Ref_FSM_BC       				 		                    *)
	(* - OUT_CU.tCU2GR.bF_Ref_FSM_BC_SetErr generieren - falls TRUE wird der Backupwert (Parameter) verwendet*)
	OUT_CU.tCU2GR.rF_Ref_FSM_BC;      (* bus: scaling value for Reference Frequency FSM/LFSM from EU [%]	*)
	OUT_CU.tCU2GR.bF_Ref_FSM_BC_SetErr;   (* Reference Frequency FSM/LFSM measuring signal failure*)
	(********************************************************************************************)
	(************************* Control bit for blocking module***********************************)
	OUT_CU.tCU2GR.bCheck_CU2GR := IN_CU.tHA2CU.bCheck_HA2CU AND IN_CU.tGR2CU.bCheck_GR2CU;
	(********************************************************************************************)
	(********************************************************************************************)

	(********************************************************************************************)
	(************** ILF - I n t e g r a l  L o c a l  F r e q u e n c y *************************)
	(********************************************************************************************)
	(*(DE)Activating  - HW --> To connect or to set fix value    		         			    *)
	OUT_CU.bILF_SetCOn	:= IN_CU.tSet_ILF_COn.Di; 					(* DI: ILF - on (activate)	*)
	OUT_CU.bILF_SetCOf	:= IN_CU.tSet_ILF_COf.Di := TRUE; 		 (* DI: ILF - off (deactivate)	*)
	(*																							*)
	(*(DE)Activating - bus																		*)
	OUT_CU.bSet_ILF_COn_Bus; 									   (* bus: ILF - on (activate)	*)
	OUT_CU.bSet_ILF_COf_Bus	:= TRUE; 						    (* bus: ILF - off (deactivate)  *)

	(*- - - - - - - - - - - F E E D B A C K  S I G N A L S  - - - - - - - - - - - - - -- - - -  *)
	IN_CU.tILF_SOn.Do;								(*  ILF is on								*)
	IN_CU.tILF_SOf.Do;    							(*  ILF is off								*)
	(********************************************************************************************)

END_PROGRAM
```

### Program Logical/Customized/c_statGR_TC2 (IEC, version 4.09.0) - customization task for protection test

#### c_statGR_TC2Cyclic.st
```iecst
(*********************************************************************************************
AGGR: static GridCode - custom task (cyclic)

This code is confidential and proprietary to the INNIO Company.
It may not be used in any form, or reproduced in any manner, without the express
written permission of the INNIO Company.
Copyright, INNIO Company, 2019

- customized modification for generator protection

Customized modifications: -
------------------------

History:
-------
V4.09.0 28.11.2019	lettenb.  partly moved from task c_statGR for cycle time optimizing

Instructions for use:
--------------------
-
Outstandings:
-------------
*********************************************************************************************)

PROGRAM _CYCLIC

	(********************************************************************************************)
	(************************* protection test **************************************************)
	(********************************************************************************************)
    (* Protection Test 1 *)
    OUT_CU.tProtectionTest[1].Do := NOT   ((IN_CU.bMsg2801Set AND 	  IN_CU.bMMD_BB_AlarmTestOn)
										OR (IN_CU.bMsg1038Set AND NOT IN_CU.bMMD_BB_AlarmTestOn)
										OR (IN_CU.bMsg1143Set AND NOT IN_CU.bMMD_BB_AlarmTestOn)
										OR (IN_CU.bMsg1144Set AND NOT IN_CU.bMMD_BB_AlarmTestOn));

    (* Protection Test 2 *)
	OUT_CU.tProtectionTest[2].Do := NOT    (IN_CU.bMsg1109Set
	 									OR 	IN_CU.bMsg1110Set
										OR  IN_CU.bMsg1111Set
										OR  IN_CU.bMsg1126Set
										OR  IN_CU.bMsg1127Set
										OR  IN_CU.bMsg2277Set
										OR  IN_CU.bMsg2316Set);

	(* Protection Test 3 *)
	OUT_CU.tProtectionTest[3].Do := NOT   ((IN_CU.bMsg2934Set AND 	  IN_CU.bMMD_BB_AlarmTestOn)
										OR (IN_CU.bMsg1041Set AND NOT IN_CU.bMMD_BB_AlarmTestOn)
										OR (IN_CU.bMsg1042Set AND NOT IN_CU.bMMD_BB_AlarmTestOn)
										OR (IN_CU.bMsg1112Set AND NOT IN_CU.bMMD_BB_AlarmTestOn));

	(* block OUT_OP.tRel_Sync_Load.Do *)
	xTOF_Bloc_SY_ProtTest(IN:= NOT OUT_CU.tProtectionTest[1].Do OR NOT OUT_CU.tProtectionTest[2].Do OR NOT OUT_CU.tProtectionTest[3].Do, PT := T#1s);
	OUT_CU.bBloc_SY_ProtTest := xTOF_Bloc_SY_ProtTest.Q;

END_PROGRAM
```

#### c_statGR_TC2Init.st
```iecst
PROGRAM _INIT

(* TODO : Add your code here *)

END_PROGRAM
```

#### c_statGR_TC2.var
```iecst
VAR
	xTOF_Bloc_SY_ProtTest : TOF;
END_VAR

VAR CONSTANT

END_VAR
```

### Program Logical/Customized/c_fc (IEC, version 4.13.0) - customisation task for frequency control
